// TIA Portal V16 export
// export: Created 2025-08-01T13:37:59.2816162Z, ExportSetting WithDefaults, DisplayName Totally Integrated Automation Portal, DisplayVersion V16, DisplayName TIA Portal Version Control Interface, DisplayVersion V16, DisplayName TIA Portal Openness, DisplayVersion V16, DisplayName STEP 7 Professional, DisplayVersion V16, DisplayName STEP 7 Safety, DisplayVersion V16, DisplayName WinCC Advanced, DisplayVersion V16
FUNCTION_BLOCK "DriveConfirmation_Function"   // FB5, FBD
TITLE = Drive Confirmation Function Block
VERSION : 0.1
// stored: AutoNumber true, IsIECCheckEnabled false, UDAEnableTagReadback false
   VAR_INPUT
      "System RUN" : Bool;
      "Drive Ouput Q" : Bool;
      "Drive Ready Signal" : Bool;
      DelayTime : Time := T#1s;
   END_VAR
   VAR_OUTPUT
      "Timer ET" : Time;
      "Ouput WORD" : Bool;
   END_VAR
BEGIN

REGION Network 1: Confirmation Drive
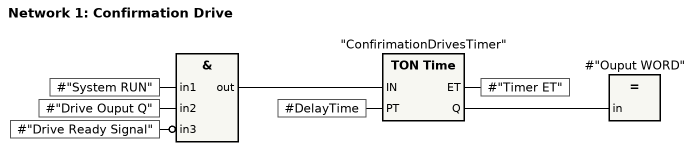
   "ConfirimationDrivesTimer".TON(IN := #"System RUN" AND #"Drive Ouput Q" AND NOT #"Drive Ready Signal",
                           PT := #DelayTime,
                           ET => #"Timer ET");
   #"Ouput WORD" := "ConfirimationDrivesTimer".Q;
END_REGION
END_FUNCTION_BLOCK
